FUNCTION_BLOCK Technology EXTENDS TcoCore.TcoContext
VAR
    _processSettings : ProcessDataManager(THIS^);
    _cu00x           : CU00x(THIS^);
END_VAR

(*~
	<docu>
		<summary>
			Main method of the TcoContext. This is the entry point of any control logic that belongs to this context. 
			The call of this method is ensured by calling the <c>InstanceName.Run()</c> method, and it must not be called explicitly.
			This method is abstract, and it must be overridden in derived block.
		</summary>
	</docu>
~*)
METHOD PROTECTED  Main
_cu00x();
END_METHOD

PROPERTY ProcessSettings : REFERENCE TO ProcessDataManager
GET
ProcessSettings REF= _processSettings;
END_GET
END_PROPERTY

END_FUNCTION_BLOCK

(* stored: Version 1.1.0.1, ProductVersion 3.1.4024.9
   POU Technology: Id {20d051ba-8e3a-4d8b-9fb7-71f6957f3a63}, SpecialFunc None
   Method Main: Id {d1d0e200-21d1-4642-b4c8-2fd801b60f39}
   Property ProcessSettings: Id {5f876a71-a280-42cf-9f33-fc8ef671f9a2}
   Get Get: Id {4cb3435a-d869-4802-9d86-6466a1c918f7} *)
